FUNCTION_BLOCK FB_HE_SATT_FilterCombinationToTransmission
VAR
END_VAR

END_FUNCTION_BLOCK

(* stored: Version 1.1.0.1
   POU FB_HE_SATT_FilterCombinationToTransmission: Id {57b92a13-f75a-4ff7-bbe9-5e6dee3c26e5}, SpecialFunc None *)
